// LS Electric XG5000 project: 0122 16진수
// PLC LSPLC

PROGRAM NewProgram (task: 스캔 프로그램)

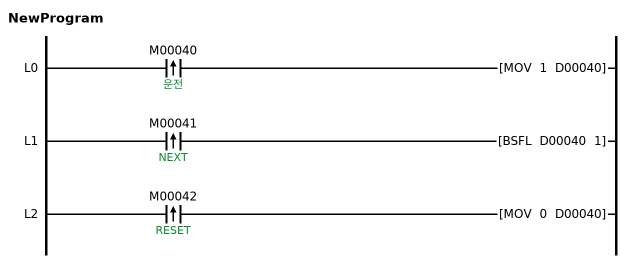
; L0
LOADP     M00040	// 운전
MOV       1 D00040
; L1
LOADP     M00041	// NEXT
BSFL      D00040 1
; L2
LOADP     M00042	// RESET
MOV       0 D00040